{attribute 'linkalways'} 
{attribute 'no_explicit_call' := 'This FB is a CLASS and must be accessed using methods or properties'}
{attribute 'enable_dynamic_creation'}
FUNCTION_BLOCK _ETcVnKeypointDetectionTypeAGAST EXTENDS EnumDatatypeBase
VAR
	localData : ETcVnKeypointDetectionTypeAGAST;
	activeData : REFERENCE TO ETcVnKeypointDetectionTypeAGAST;
	enumBaseDatatype : _DINT(localData);
END_VAR

METHOD PRIVATE AddLocalEnumeration
VAR_INPUT
	Enumeration : T_MAXSTRING;
	Value : ETcVnKeypointDetectionTypeAGAST;
END_VAR
AddEnumeration(Enumeration, Value);
END_METHOD

PROPERTY PUBLIC Address : PVOID
GET
Address := ADR(activeData);
END_GET
END_PROPERTY

METHOD PUBLIC ClearReference
VAR_INPUT
END_VAR
activeData REF= localData;
SetBaseDatatypeReference();
END_METHOD

METHOD PUBLIC Clone : I_Datatype
VAR
    pClone : POINTER TO _ETcVnKeypointDetectionTypeAGAST;
END_VAR
pClone := __NEW(_ETcVnKeypointDetectionTypeAGAST(InitialValue := Value));
Clone := pClone^;
END_METHOD

METHOD FB_init : BOOL
VAR_INPUT
	bInitRetains : BOOL; // if TRUE, the retain variables are initialized (warm start / cold start)
	bInCopyCode : BOOL;  // if TRUE, the instance afterwards gets moved into the copy code (online change)
	InitialValue : ETcVnKeypointDetectionTypeAGAST;
END_VAR
localData := InitialValue;
AddBaseDatatype(enumBaseDatatype);
ClearReference();

AddLocalEnumeration('TCVN_KDT_AGAST_5_8', ETcVnKeypointDetectionTypeAGAST.TCVN_KDT_AGAST_5_8);
AddLocalEnumeration('TCVN_KDT_AGAST_7_12d', ETcVnKeypointDetectionTypeAGAST.TCVN_KDT_AGAST_7_12d);
AddLocalEnumeration('TCVN_KDT_AGAST_7_12s', ETcVnKeypointDetectionTypeAGAST.TCVN_KDT_AGAST_7_12s);
AddLocalEnumeration('TCVN_KDT_AGAST_9_16', ETcVnKeypointDetectionTypeAGAST.TCVN_KDT_AGAST_9_16);
END_METHOD

PROPERTY PUBLIC Identifier : T_MAXSTRING
GET
Identifier := 'ETcVnKeypointDetectionTypeAGAST';
END_GET
END_PROPERTY

METHOD IsEnumeratorValueEqual : BOOL
VAR_INPUT
	Enumerator : I_KeyValueForwardEnumerator;
END_VAR
VAR
	storedValue : ETcVnKeypointDetectionTypeAGAST;
END_VAR
IF NOT Enumerator.TryGet(storedValue) THEN
	RETURN;
END_IF

IsEnumeratorValueEqual := storedValue = activeData;
END_METHOD

METHOD PUBLIC MakeReferenceTo
VAR_INPUT
	ReferenceTarget : REFERENCE TO ETcVnKeypointDetectionTypeAGAST;
END_VAR
activeData REF= ReferenceTarget;
SetBaseDatatypeReference();
END_METHOD

METHOD PROTECTED SetBaseDatatypeReference
VAR_INPUT
END_VAR
enumBaseDatatype.MakeReferenceTo(activeData);
END_METHOD

PROPERTY PUBLIC Size : UDINT
GET
Size := SIZEOF(activeData);
END_GET
END_PROPERTY

METHOD TryMakeReferenceTo : BOOL
VAR_INPUT
	Target : I_Datatype;
END_VAR
VAR
	targetAsEnum : I_EnumDatatype;
	pTargetData : POINTER TO ETcVnKeypointDetectionTypeAGAST;
END_VAR
IF NOT Target.TryResolveAsEnumDatatype(targetAsEnum) THEN
	RETURN;
END_IF

IF targetAsEnum.Identifier <> Identifier THEN
	RETURN;
END_IF

pTargetData := Target.Address;
activeData REF= pTargetData^;
SetBaseDatatypeReference();
TryMakeReferenceTo := TRUE;
END_METHOD

PROPERTY PUBLIC Value : ETcVnKeypointDetectionTypeAGAST
GET
Value := activeData;
END_GET
SET
activeData := Value;
END_SET
END_PROPERTY

END_FUNCTION_BLOCK

(* stored: Version 1.1.0.1
   POU _ETcVnKeypointDetectionTypeAGAST: Id {46aa8f7f-8e8e-46cb-ae7f-81d1cb175bc5}, SpecialFunc None
   Folder Constructor: Id {b9c124df-a1c6-4d96-b430-83c3185b0f39}
   Folder Private: Id {a9fc6e5f-bc13-423b-b8fc-7f1f63950245}
   Folder Protected: Id {f7b79c9b-85d2-4644-8e06-7143ca3b7d4d}
   Method AddLocalEnumeration: Id {a3f64c2c-7dc8-453b-8660-5a5525baa955}
   Property Address: Id {3e9ea633-94c1-4008-9ced-19d431bbbb00}
   Get Get: Id {7188e831-5222-44e4-b7fc-fa460673b8ac}
   Method ClearReference: Id {e99b539f-0628-429d-a94e-91f29024f62a}
   Method Clone: Id {9d3acf34-f8ed-4646-9bb0-377d61655054}
   Method FB_init: Id {4a1e1f5a-dd1e-4b59-8569-944016a8f2c7}
   Property Identifier: Id {7ae25151-3d34-48bf-8ccd-0cd0eb7cc7bf}
   Get Get: Id {408e65d3-d9b5-437d-a4c3-87cb57ddb723}
   Method IsEnumeratorValueEqual: Id {80a5693b-c876-4d1c-83ee-d5d00f8032da}
   Method MakeReferenceTo: Id {ba35d24a-ea4b-417b-bc27-4c145cc27aa8}
   Method SetBaseDatatypeReference: Id {b2c8664e-7020-4ab7-a26c-d6f5abde9491}
   Property Size: Id {65b9d827-6d08-4978-afd7-3d4e479db718}
   Get Get: Id {5c43146e-2033-4b59-966c-d336032ac7f6}
   Method TryMakeReferenceTo: Id {6fab3bfc-f239-440d-8b96-72a12602d751}
   Property Value: Id {e701de79-eda5-4a14-bb08-fec1abf8c818}
   Get Get: Id {80a4790e-1efb-4b87-b5af-24560c6534b2}
   Set Set: Id {32da9933-caf7-46ac-a38b-56774e04050c} *)
